SUBAPPLICATION Ventilsteuerung_Uebung_003 (* DigitalInput_I1/_I2 auf DigitalOutput_Q1/_I2 *)
  (* Standard: 61499-2 *)
  (* Version 1.0, 2023-10-23, franz *)
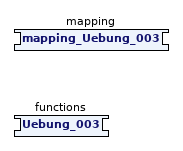
  SUBAPPS
    mapping : mapping_Uebung_003;
    functions : Uebung_003;
  END_SUBAPPS
END_SUBAPPLICATION
